TYPE PanelButton :
STRUCT
	alias   : STRING;
	pressed : BOOL;
	row   	: INT;
	column 	: INT;
END_STRUCT
END_TYPE

(* stored: Version 1.1.0.1
   DUT PanelButton: Id {821dd715-1078-4fbb-ba7b-9326cd27a5b0} *)
